{attribute 'hide_all_locals'}
FUNCTION_BLOCK TraceMessageInfo IMPLEMENTS I_TraceMessageInfo
VAR
	_Message   : T_MaxString;
	_MessageId : UDINT;
	_Severity  : USINT;
END_VAR

{attribute 'monitoring':='call'}
PROPERTY Message : T_MaxString
GET
Message := _Message;
END_GET
SET
_Message := Message;
END_SET
END_PROPERTY

{attribute 'monitoring':='call'}
PROPERTY MessageId : UDINT
GET
MessageId := _MessageId;
END_GET
SET
_MessageId := MessageId;
END_SET
END_PROPERTY

{attribute 'monitoring':='call'}
PROPERTY Severity : USINT
GET
Severity := _Severity;
END_GET
SET
_Severity := Severity;
END_SET
END_PROPERTY

END_FUNCTION_BLOCK

(* stored: Version 1.1.0.1, ProductVersion 3.1.4026.18
   POU TraceMessageInfo: Id {0a4ff03a-775d-4fc4-ad9a-908d10a0b53e}, SpecialFunc None
   Property Message: Id {d8ad990d-197a-4267-99ed-b778584f8c85}
   Get Get: Id {eb64778f-b4d1-44d8-ab14-4f75fec28446}
   Set Set: Id {2590b935-9ec1-4c88-ba94-97649951e8b3}
   Property MessageId: Id {4b607a47-3840-4b8c-a68f-324d0b00851e}
   Get Get: Id {0b9a68a8-6345-4777-a64c-de076e04b7a7}
   Set Set: Id {b4feef98-4a2a-4ea1-bf46-e1f86817b493}
   Property Severity: Id {c5732040-1b0d-416f-99fa-94f79ffe2339}
   Get Get: Id {4466334a-70d2-4e42-8fe6-82e3024d775a}
   Set Set: Id {a7b60124-ff24-4666-9609-de024f1498b4} *)
